// TwinCAT 3 PLC project Tc_SortingStation
// ProgramVersion: 3.1.4024.0
// libraries:
//   PlantControl and CMs, * (ArmAutomation)
//   Tc2_Standard, * (Beckhoff Automation GmbH)
//   Tc2_System, * (Beckhoff Automation GmbH)
//   Tc3_Module, * (Beckhoff Automation GmbH)
// project tree:
//   DUTs/ CM_DIN_UDT.TcDUT, CM_DO_UDT.TcDUT, CM_Vision_UDT.TcDUT
//   GVLs/ FIO.TcGVL, GVL.TcGVL
//   / PlcTask.TcTTO
//   POUs/ControlModules/ CM_DIN.TcPOU, CM_DO.TcPOU, CM_VisionSensor.TcPOU
//   POUs/EquipmentModules/FBD/ FB_ConveyorEntry_FBD.TcPOU
//   POUs/EquipmentModules/LAD/ FB_Conveyor.TcPOU, FB_Sorter.TcPOU
//   POUs/EquipmentModules/ST/ FB_ConveyorEntry_ST.TcPOU, FB_ConveyorExit_ST.TcPOU
//   POUs/ MAIN.TcPOU
// real-time tasks:
//   TASK PlcTask: cycle T#10ms, priority 20, ADS port 350

CONFIGURATION Tc_SortingStation
    RESOURCE PLC ON TwinCAT3
        TASK PlcTask(INTERVAL := T#10ms, PRIORITY := 20);
        PROGRAM MAIN WITH PlcTask : MAIN;
    END_RESOURCE
END_CONFIGURATION

// ---- DUTs/CM_DIN_UDT.TcDUT
TYPE CM_DIN_UDT :
STRUCT
	SensorInput : BOOL;
	
	AutoHigh : BOOL;
END_STRUCT
END_TYPE

// ---- DUTs/CM_DO_UDT.TcDUT
TYPE CM_DO_UDT :
STRUCT
	PI_Enable : BOOL;
	
	PO_HighCommand : BOOL;
	PO_LowCommand : BOOL;
END_STRUCT
END_TYPE

// ---- DUTs/CM_Vision_UDT.TcDUT
TYPE CM_Vision_UDT :
STRUCT
	Input : DINT;
	
	PO_PV : DINT;
END_STRUCT
END_TYPE

// ---- GVLs/FIO.TcGVL
{attribute 'qualified_only'}
VAR_GLOBAL

//Sensor	Bool	FACTORY I/O (Running)	496	FALSE
//Sensor	Bool	FACTORY I/O (Paused)	497	FALSE
//Sensor	Bool	FACTORY I/O (Reset)	498	FALSE
bAtExit : BOOL;	//Sensor	Bool	At exit	2	TRUE

//bEmgStop : BOOL; //Sensor	Bool	Emergency stop	0	TRUE
//bStart : BOOL;	//Sensor	Bool	Start	1	FALSE
//bStop : BOOL;	//Sensor	Bool	Stop	3	TRUE
//bReset : BOOL;	//Sensor	Bool	Reset	4	FALSE
//bManual : BOOL;	//Sensor	Bool	Manual	5	TRUE
//bAuto : BOOL; 	//Sensor	Bool	Auto	6	FALSE

//Sensor	Float	FACTORY I/O (Time Scale)	240	0
iVisionSensor : DINT;	//Sensor	Int	Vision sensor	0	0
//Actuator	Bool	FACTORY I/O (Run)	496	FALSE
//Actuator	Bool	FACTORY I/O (Pause)	497	FALSE
//Actuator	Bool	FACTORY I/O (Reset)	498	FALSE
bEmitter : BOOL; //Actuator	Bool	Emitter	0	TRUE
bConveyorEntry_out: BOOL; 	//Actuator	Bool	Entry conveyor	1	FALSE
bConveyorExit_out : BOOL; 		//Actuator	Bool	Exit conveyor	2	FALSE
bStopBlade : BOOL; 	//Actuator	Bool	Stop blade	3	FALSE
//Actuator	Bool	-	6	FALSE
bSorter_1_out : BOOL;	//Actuator	Bool	Sorter 1 belt	5	FALSE
bSorter_1_turn : BOOL;	//Actuator	Bool	Sorter 1 turn	4	FALSE
//Actuator	Bool	-	9	FALSE
bSorter_2_out : BOOL;	//Actuator	Bool	Sorter 2 belt	8	FALSE
bSorter_2_turn : BOOL;	//Actuator	Bool	Sorter 2 turn	7	FALSE
//Actuator	Bool	-	12	FALSE
bSorter_3_out : BOOL;	//Actuator	Bool	Sorter 3 belt	11	FALSE
bSorter_3_turn : BOOL;	//Actuator	Bool	Sorter 3 turn	10	FALSE
//Actuator	Bool	Remover 1	13	TRUE
//Actuator	Bool	Remover 2	14	TRUE
//Actuator	Bool	Remover 3	15	TRUE
//Actuator	Bool	Start light	16	FALSE
//Actuator	Bool	Stop light	17	FALSE
//Actuator	Bool	Reset light	18	FALSE
//Actuator	Int	FACTORY I/O (Camera Position)	240	0
//Actuator	Int	Counter 3	2	0
//Actuator	Int	Counter 1	0	0
//Actuator	Int	Counter 2	1	0

END_VAR

// ---- GVLs/GVL.TcGVL
{attribute 'qualified_only'}
VAR_GLOBAL
	GREEN_BOTTOM : BOOL; // 4
	GREEN_TOP : BOOL;	// 5
	GREEN_MIDDLE : BOOL; // 6
	
	BLUE_BOTTOM : BOOL; // 1
	BLUE_TOP : BOOL; // 2
	BLUE_MIDDLE : BOOL; // 3
	
	SortingDone : BOOL;
	readyForSorting : BOOL;
END_VAR

// ---- POUs/MAIN.TcPOU
PROGRAM MAIN
VAR
	
	//FBs
	fbPlantControl : PlantAndCMs.FB_PlantControl_mode_1;
	Ctrl_data_Plant : PlantAndCMs.Udt_PlantControl_Mode_1;
	
	//Equipment modules structured IN LADDER
	LAD_fbConveyorEntry : FB_Conveyor;
	LAD_fbSorter : FB_Sorter;
	
	//Equipment modules structured in ST
	ST_fbConveyorEntry : FB_ConveyorEntry_ST;
	ST_fbConveyorExit : FB_ConveyorExit_ST;
	
	// Control modules call
	cmVision : CM_VisionSensor;
	Ctrl_data_vision : CM_Vision_UDT;
	
	cmConveyor1 : CM_DO;
	cmConveyor2 : CM_DO;
	Ctrl_data_Conveyor1 : CM_DO_UDT;
	Ctrl_data_Conveyor2 : CM_DO_UDT;
	
	cmAtExit : CM_DIN;
	Ctrl_data_exit : CM_DIN_UDT;
	
	cmSorter1 : CM_DO;
	Crtl_data_sorter1 : CM_DO_UDT;
	cmSorter2 : CM_DO;
	Crtl_data_sorter2 : CM_DO_UDT;
	cmSorter3 : CM_DO;
	Crtl_data_sorter3 : CM_DO_UDT;
	
	cmStopBlade : CM_DO;
	crtl_data_StopBlade : CM_DO_UDT;
	
	cmEmitter : CM_DO;
	ctrl_data_emitter : CM_DO_UDT;
	
END_VAR

VAR_IN_OUT
	
END_VAR



fbPlantControl(
	on_in := TRUE,
	Auto_In := PlantAndCMs.FIO.bAuto,
	Manual_In := PlantAndCMs.FIO.bManual,
	
	EmgStop_In := PlantAndCMs.FIO.bEmgStop,
	Start_In := PlantAndCMs.FIO.bStart,
	Stop_In := PlantAndCMs.FIO.bStop, 
	Reset_In := PlantAndCMs.FIO.bReset,
	
	Ctrl_Plant := Ctrl_data_Plant
);
	

LAD_fbConveyorEntry(
		control_data := Ctrl_data_plant,
		
		control_data_vision := Ctrl_data_vision,
		control_data_Conveyor1 := Ctrl_data_Conveyor1,
		control_data_StopBlade := crtl_data_StopBlade,
		control_data_emitter := ctrl_data_emitter
		);	
	
LAD_fbSorter(
		control_data := Ctrl_data_plant,
		control_data_vision := Ctrl_data_vision,
		control_data_Conveyor2 := Ctrl_data_Conveyor2,
		control_data_sorter1 := Crtl_data_sorter1,
		control_data_sorter2 := Crtl_data_sorter2,
		control_data_sorter3 := Crtl_data_sorter3,
		control_data_atExit := Ctrl_data_exit,
	
	);	

(*
ST_fbConveyorEntry(
		control_data := Ctrl_data_plant,
		
		control_data_vision := Ctrl_data_vision,
		control_data_Conveyor1 := Ctrl_data_Conveyor1,
		control_data_StopBlade := crtl_data_StopBlade,
		control_data_emitter := ctrl_data_emitter
		);	

ST_fbConveyorExit(
		control_data := Ctrl_data_plant,
		control_data_vision := Ctrl_data_vision,
		control_data_Conveyor2 := Ctrl_data_Conveyor2,
		control_data_sorter1 := Crtl_data_sorter1,
		control_data_sorter2 := Crtl_data_sorter2,
		control_data_sorter3 := Crtl_data_sorter3,
		control_data_atExit := Ctrl_data_exit
		);
*)
		

//// CM Calls
cmConveyor1( 
	Control_data_DO := Ctrl_data_Conveyor1,
	
   	PO_HighCommand => FIO.bConveyorEntry_out
	); 
 
cmConveyor2(
	Control_data_DO := Ctrl_data_Conveyor2,
	PO_HighCommand => FIO.bConveyorExit_out
	);
	
cmAtExit(
	PI_autoHigh := FIO.bAtExit,
	Control_data := Ctrl_data_exit);

	
cmVision(
	SensorInput := FIO.iVisionSensor,
	control_data_vision := Ctrl_data_Vision);
	
cmSorter1(
	Control_data_DO := Crtl_data_sorter1,
	PO_HighCommand => FIO.bSorter_1_out, 
	PO_HighCommand => FIO.bSorter_1_turn
	);
cmSorter2(
	Control_data_DO := Crtl_data_sorter2,
	PO_HighCommand => FIO.bSorter_2_out, 
	PO_HighCommand => FIO.bSorter_2_turn
	);
	
cmSorter3(
	Control_data_DO := Crtl_data_sorter3,
	PO_HighCommand => FIO.bSorter_3_out,
	PO_HighCommand => FIO.bSorter_3_turn
	);
	
cmStopBlade(
	Control_data_DO := crtl_data_StopBlade,
	PO_HighCommand => FIO.bStopBlade
	);
cmEmitter(
	PO_HighCommand => FIO.bEmitter,
	Control_data_DO := ctrl_data_emitter
	);

END_PROGRAM

// ---- POUs/EquipmentModules/LAD/FB_Conveyor.TcPOU
FUNCTION_BLOCK FB_Conveyor
VAR_INPUT
	
END_VAR
VAR_OUTPUT
END_VAR
VAR
	on : BOOL;
	timer0_emitter : Tc2_Standard.TP;
	EmitterTrigger : BOOL;
	Timer1 : Tc2_Standard.TON;
	Step_0_Standby : BOOL;
	Step_1 : BOOL;
	Step_2 : BOOL;
	Step_3 : BOOL;
	Step_4 : BOOL;
	Step_5 : BOOL;
	Step_6 : BOOL;
	Step_7 : BOOL;
	Step_10 : BOOL;
	Step_15 : BOOL;
	step_last : BOOL;
	
	condition : BOOL;
	
	Opstart_puls_OS : BOOL;

	
	Initialiser_SQ: BOOL;
END_VAR
VAR_IN_OUT
	control_data : PlantAndCMs.Udt_PlantControl_Mode_1;
	
	control_data_vision : CM_Vision_UDT;
	control_data_Conveyor1 : CM_DO_UDT;
	
	control_data_StopBlade : CM_DO_UDT;
	control_data_emitter : CM_DO_UDT;
END_VAR
VAR // added by the converter: edge detectors and wires of the graphical bodies
    _w1, _w2, _w3, _w4, _w5, _w6, _w7, _w8, _w9, _w10, _w11, _w12, _w13, _w14, _w15, _w16, _w17 : BOOL;
END_VAR

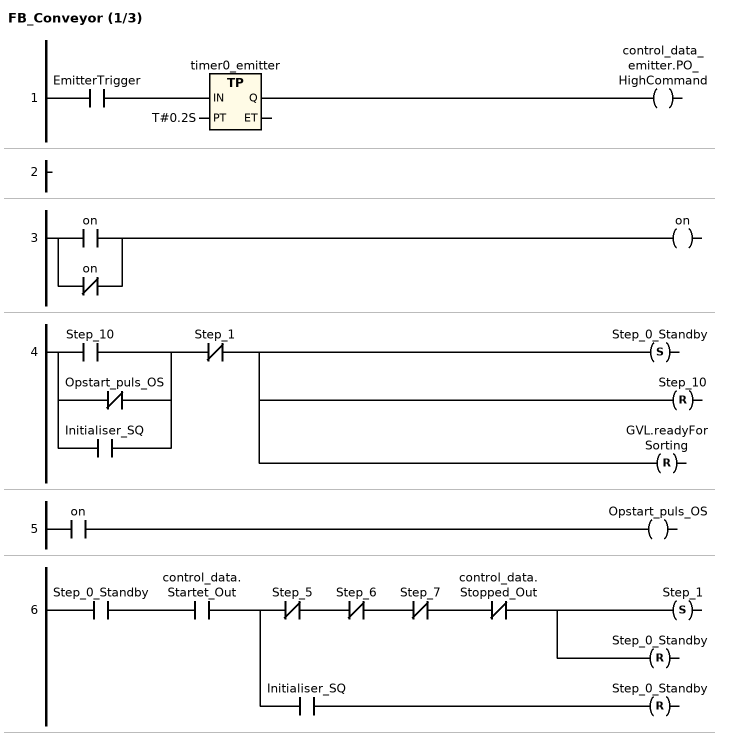
// NETWORK 1
timer0_emitter(IN := EmitterTrigger, PT := T#0.2S); // TP
control_data_emitter.PO_HighCommand := timer0_emitter.Q;

// NETWORK 2

// NETWORK 3
on := on OR NOT on;

// NETWORK 4
_w1 := (Step_10 OR NOT Opstart_puls_OS OR Initialiser_SQ) AND NOT Step_1;
Step_0_Standby S= _w1;
Step_10 R= _w1;
GVL.readyForSorting R= _w1;

// NETWORK 5
Opstart_puls_OS := on;

// NETWORK 6
_w2 := Step_0_Standby AND control_data.Startet_Out;
_w3 := _w2 AND NOT Step_5 AND NOT Step_6 AND NOT Step_7 AND NOT control_data.Stopped_Out;
Step_1 S= _w3;
Step_0_Standby R= _w3;
Step_0_Standby R= _w2 AND Initialiser_SQ;

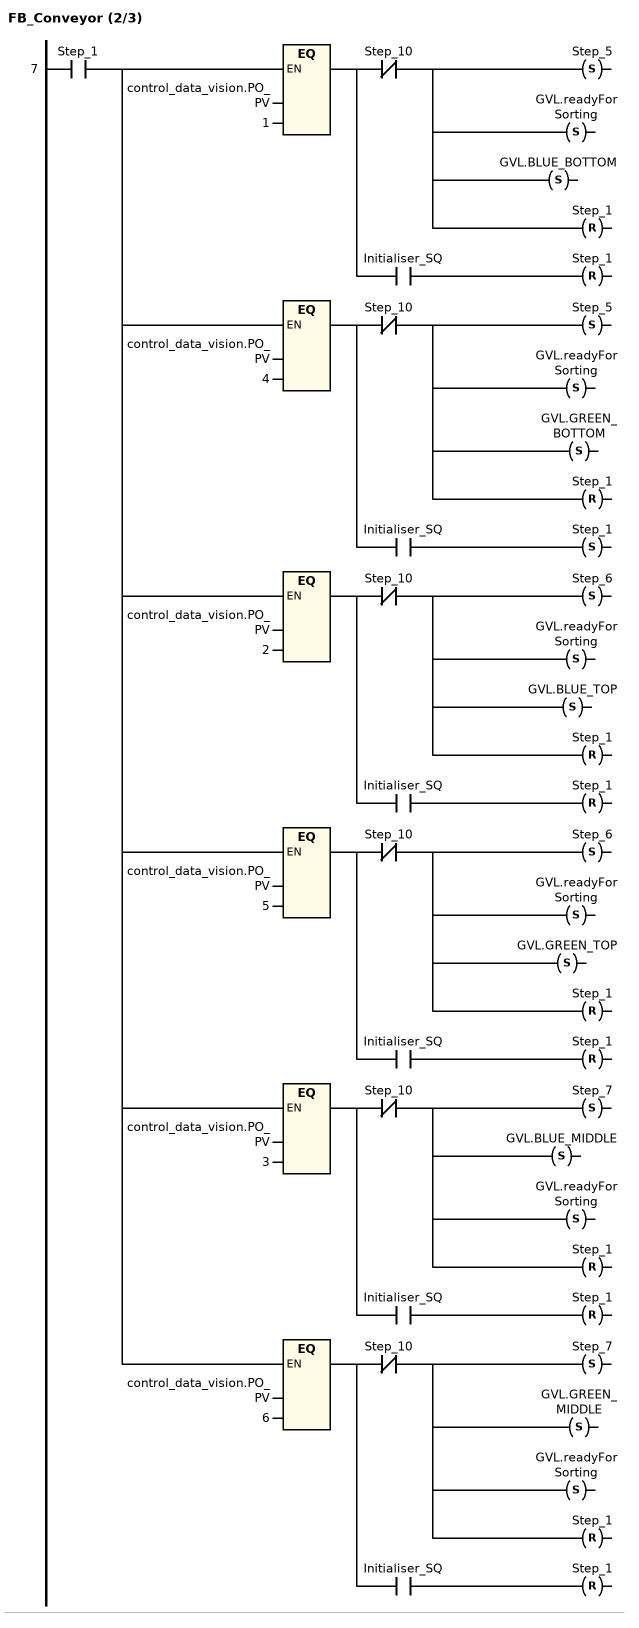
// NETWORK 7
_w4 := Step_1;
_w5 := _w4 AND control_data_vision.PO_PV = 1;
_w6 := _w5 AND NOT Step_10;
Step_5 S= _w6;
GVL.readyForSorting S= _w6;
GVL.BLUE_BOTTOM S= _w6;
Step_1 R= _w6;
Step_1 R= _w5 AND Initialiser_SQ;
_w7 := _w4 AND control_data_vision.PO_PV = 4;
_w8 := _w7 AND NOT Step_10;
Step_5 S= _w8;
GVL.readyForSorting S= _w8;
GVL.GREEN_BOTTOM S= _w8;
Step_1 R= _w8;
Step_1 S= _w7 AND Initialiser_SQ;
_w9 := _w4 AND control_data_vision.PO_PV = 2;
_w10 := _w9 AND NOT Step_10;
Step_6 S= _w10;
GVL.readyForSorting S= _w10;
GVL.BLUE_TOP S= _w10;
Step_1 R= _w10;
Step_1 R= _w9 AND Initialiser_SQ;
_w11 := _w4 AND control_data_vision.PO_PV = 5;
_w12 := _w11 AND NOT Step_10;
Step_6 S= _w12;
GVL.readyForSorting S= _w12;
GVL.GREEN_TOP S= _w12;
Step_1 R= _w12;
Step_1 R= _w11 AND Initialiser_SQ;
_w13 := _w4 AND control_data_vision.PO_PV = 3;
_w14 := _w13 AND NOT Step_10;
Step_7 S= _w14;
GVL.BLUE_MIDDLE S= _w14;
GVL.readyForSorting S= _w14;
Step_1 R= _w14;
Step_1 R= _w13 AND Initialiser_SQ;
_w15 := _w4 AND control_data_vision.PO_PV = 6;
_w16 := _w15 AND NOT Step_10;
Step_7 S= _w16;
GVL.GREEN_MIDDLE S= _w16;
GVL.readyForSorting S= _w16;
Step_1 R= _w16;
Step_1 R= _w15 AND Initialiser_SQ;

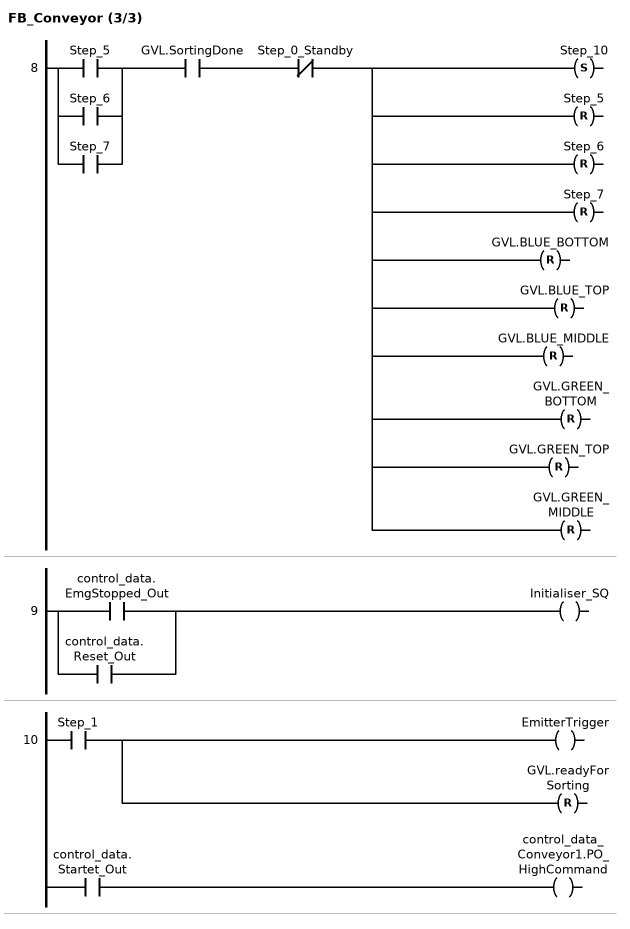
// NETWORK 8
_w17 := (Step_5 OR Step_6 OR Step_7) AND GVL.SortingDone AND NOT Step_0_Standby;
Step_10 S= _w17;
Step_5 R= _w17;
Step_6 R= _w17;
Step_7 R= _w17;
GVL.BLUE_BOTTOM R= _w17;
GVL.BLUE_TOP R= _w17;
GVL.BLUE_MIDDLE R= _w17;
GVL.GREEN_BOTTOM R= _w17;
GVL.GREEN_TOP R= _w17;
GVL.GREEN_MIDDLE R= _w17;

// NETWORK 9
Initialiser_SQ := control_data.EmgStopped_Out OR control_data.Reset_Out;

// NETWORK 10
EmitterTrigger := Step_1;
GVL.readyForSorting R= Step_1;
control_data_Conveyor1.PO_HighCommand := control_data.Startet_Out;

END_FUNCTION_BLOCK

// ---- POUs/EquipmentModules/LAD/FB_Sorter.TcPOU
FUNCTION_BLOCK FB_Sorter
VAR_INPUT
END_VAR
VAR_OUTPUT
END_VAR
VAR
	on : BOOL;
	
	rTrigAtExit : Tc2_Standard.R_TRIG;
	exitTrigger : BOOL;
	atExitEdgeDetected : BOOL;
	
	Step_0_Standby : BOOL;
	Step_1 : BOOL;
	Step_2 : BOOL;
	Step_3 : BOOL;
	Step_4 : BOOL;
	Step_5 : BOOL;
	Step_6 : BOOL;
	Step_7 : BOOL;
	Step_10 : BOOL;
	Step_15 : BOOL;
	step_last : BOOL;
	
	dummy : BOOL;
	
	condition : BOOL;
	
	Opstart_puls_OS : BOOL;

	Initialiser_SQ: BOOL;
END_VAR
VAR_IN_OUT
	control_data : PlantAndCMs.Udt_PlantControl_Mode_1;
	
	control_data_vision : CM_Vision_UDT;
	control_data_Conveyor2 : CM_DO_UDT;
	
	control_data_sorter1 : CM_DO_UDT;
	control_data_sorter2 : CM_DO_UDT;
	control_data_sorter3 : CM_DO_UDT;
	
	control_data_atExit : CM_DIN_UDT;
	
	
END_VAR
VAR // added by the converter: edge detectors and wires of the graphical bodies
    _w1, _w2, _w3, _w4, _w5, _w6, _w7, _w8, _w9, _w10, _w11 : BOOL;
END_VAR

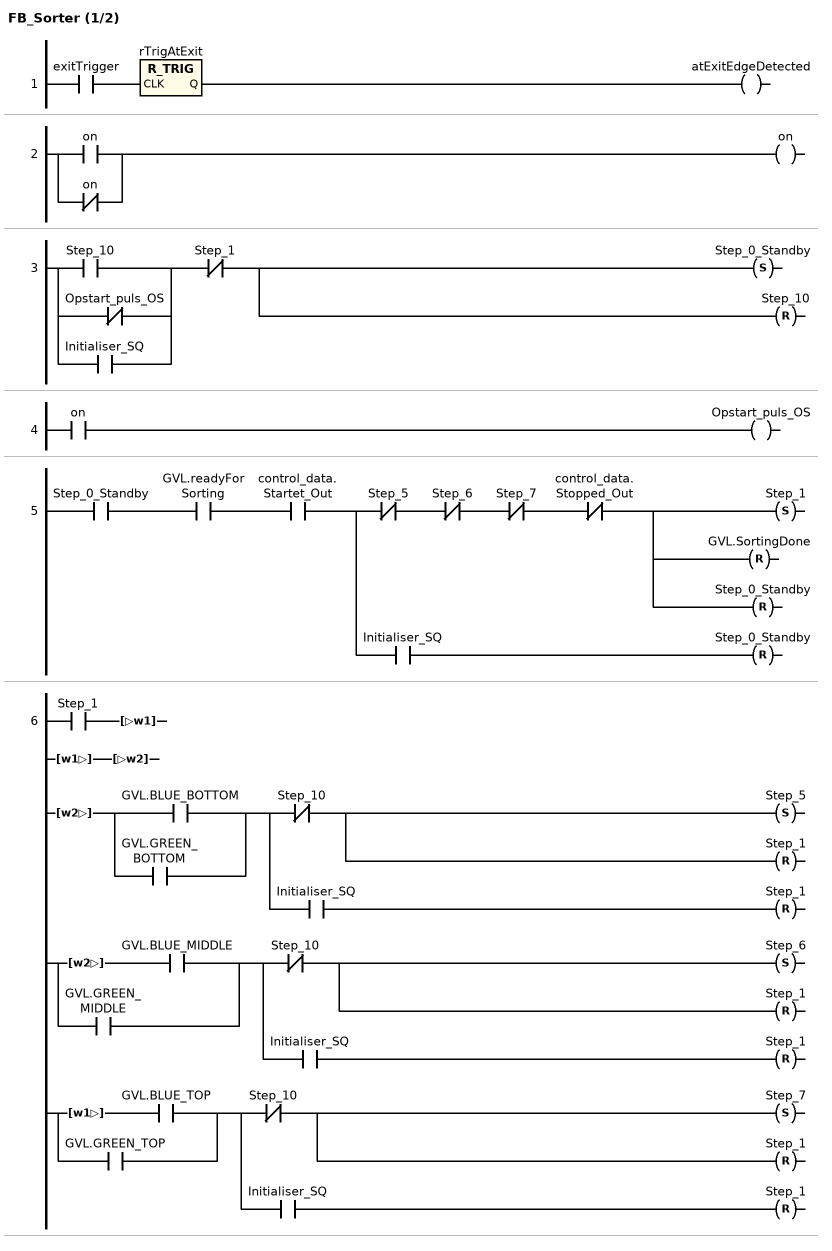
// NETWORK 1
rTrigAtExit(CLK := exitTrigger); // R_TRIG
atExitEdgeDetected := rTrigAtExit.Q;

// NETWORK 2
on := on OR NOT on;

// NETWORK 3
_w1 := (Step_10 OR NOT Opstart_puls_OS OR Initialiser_SQ) AND NOT Step_1;
Step_0_Standby S= _w1;
Step_10 R= _w1;

// NETWORK 4
Opstart_puls_OS := on;

// NETWORK 5
_w2 := Step_0_Standby AND GVL.readyForSorting AND control_data.Startet_Out;
_w3 := _w2 AND NOT Step_5 AND NOT Step_6 AND NOT Step_7 AND NOT control_data.Stopped_Out;
Step_1 S= _w3;
GVL.SortingDone R= _w3;
Step_0_Standby R= _w3;
Step_0_Standby R= _w2 AND Initialiser_SQ;

// NETWORK 6
_w4 := Step_1;
_w5 := _w4 AND (GVL.BLUE_BOTTOM OR GVL.GREEN_BOTTOM);
_w6 := _w5 AND NOT Step_10;
Step_5 S= _w6;
Step_1 R= _w6;
Step_1 R= _w5 AND Initialiser_SQ;
_w7 := _w4 AND GVL.BLUE_MIDDLE OR GVL.GREEN_MIDDLE;
_w8 := _w7 AND NOT Step_10;
Step_6 S= _w8;
Step_1 R= _w8;
Step_1 R= _w7 AND Initialiser_SQ;
_w9 := _w4 AND GVL.BLUE_TOP OR GVL.GREEN_TOP;
_w10 := _w9 AND NOT Step_10;
Step_7 S= _w10;
Step_1 R= _w10;
Step_1 R= _w9 AND Initialiser_SQ;

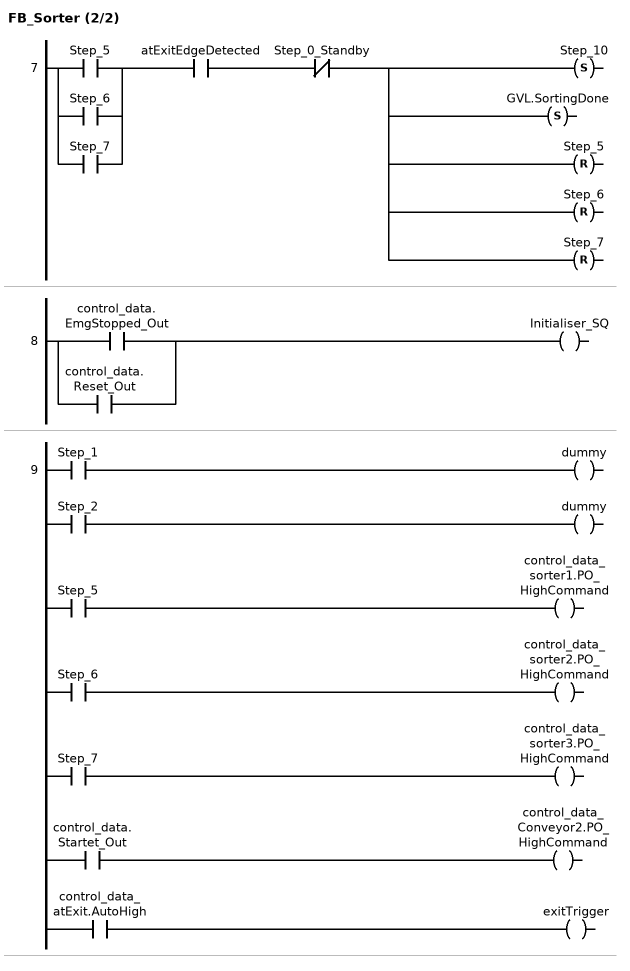
// NETWORK 7
_w11 := (Step_5 OR Step_6 OR Step_7) AND atExitEdgeDetected AND NOT Step_0_Standby;
Step_10 S= _w11;
GVL.SortingDone S= _w11;
Step_5 R= _w11;
Step_6 R= _w11;
Step_7 R= _w11;

// NETWORK 8
Initialiser_SQ := control_data.EmgStopped_Out OR control_data.Reset_Out;

// NETWORK 9
dummy := Step_1;
dummy := Step_2;
control_data_sorter1.PO_HighCommand := Step_5;
control_data_sorter2.PO_HighCommand := Step_6;
control_data_sorter3.PO_HighCommand := Step_7;
control_data_Conveyor2.PO_HighCommand := control_data.Startet_Out;
exitTrigger := control_data_atExit.AutoHigh;

END_FUNCTION_BLOCK

// ---- POUs/EquipmentModules/ST/FB_ConveyorEntry_ST.TcPOU
FUNCTION_BLOCK FB_ConveyorEntry_ST
VAR_INPUT
END_VAR
VAR_OUTPUT
END_VAR
VAR
	step : INT;
	RtrigInitTrigger : R_TRIG;
	initTrigger : BOOL := TRUE;
	
	eMitterTimer : Tc2_Standard.TP;
	startEmitting : BOOL;
	
END_VAR
VAR_IN_OUT
	control_data : PlantAndCMs.Udt_PlantControl_Mode_1;
	
	control_data_vision : CM_Vision_UDT;
	control_data_Conveyor1 : CM_DO_UDT;
	
	control_data_StopBlade : CM_DO_UDT;
	control_data_emitter : CM_DO_UDT;
END_VAR

RtrigInitTrigger(CLK :=initTrigger);

eMitterTimer(IN := StartEmitting, pt := T#0.2S);


CASE step OF 
	0 : // Init
	
		IF control_data.Auto_Out THEN
			initTrigger := FALSE;
			step := 1;
		END_IF
	
	1: // Step 1 start machine
		
		IF control_data.Startet_Out THEN
			initTrigger := TRUE;
			step := 2;
		END_IF
	2:			
		
		IF control_data_vision.PO_PV = 0 THEN
			startEmitting := TRUE;
			step := 5;
		END_IF
	
	5: 
		startEmitting := FALSE;
		GVL.readyForSorting := FALSE;
		GVL.SortingDone := FALSE;
		
		IF control_data_vision.PO_PV = 1 THEN
			GVL.BLUE_TOP := TRUE;
			GVL.BLUE_BOTTOM := FALSE;
			GVL.BLUE_MIDDLE := FALSE;
			GVL.GREEN_TOP := FALSE;
			GVL.GREEN_BOTTOM := FALSE;
			GVL.GREEN_MIDDLE := FALSE;
			step := 11;
		END_IF
		IF control_data_vision.PO_PV = 2 THEN
			GVL.BLUE_TOP := FALSE;
			GVL.BLUE_BOTTOM := TRUE;
			GVL.BLUE_MIDDLE := FALSE;
			GVL.GREEN_TOP := FALSE;
			GVL.GREEN_BOTTOM := FALSE;
			GVL.GREEN_MIDDLE := FALSE;
			step := 11;
		END_IF
		IF control_data_vision.PO_PV = 3 THEN
			GVL.BLUE_TOP := FALSE;
			GVL.BLUE_BOTTOM := FALSE;
			GVL.BLUE_MIDDLE := TRUE;
			GVL.GREEN_TOP := FALSE;
			GVL.GREEN_BOTTOM := FALSE;
			GVL.GREEN_MIDDLE := FALSE;
			step := 11;
		END_IF
		IF control_data_vision.PO_PV = 4 THEN
			GVL.BLUE_TOP := FALSE;
			GVL.BLUE_BOTTOM := FALSE;
			GVL.BLUE_MIDDLE := FALSE;
			GVL.GREEN_TOP := TRUE;
			GVL.GREEN_BOTTOM := FALSE;
			GVL.GREEN_MIDDLE := FALSE;
			step := 11;
		END_IF
		IF control_data_vision.PO_PV = 5 THEN
			GVL.BLUE_TOP := FALSE;
			GVL.BLUE_BOTTOM := FALSE;
			GVL.BLUE_MIDDLE := FALSE;
			GVL.GREEN_TOP := FALSE;
			GVL.GREEN_BOTTOM := TRUE;
			GVL.GREEN_MIDDLE := FALSE;
			step := 11;
		END_IF
		IF control_data_vision.PO_PV = 6 THEN
			GVL.BLUE_TOP := FALSE;
			GVL.BLUE_BOTTOM := FALSE;
			GVL.BLUE_MIDDLE := FALSE;
			GVL.GREEN_TOP := FALSE;
			GVL.GREEN_BOTTOM := FALSE;
			GVL.GREEN_MIDDLE := TRUE;
			step := 11;
		END_IF
		

	11:
		GVL.readyForSorting := TRUE;
		
		IF GVL.SortingDone THEN
			GVL.BLUE_TOP := FALSE;
			GVL.BLUE_BOTTOM := FALSE;
			GVL.BLUE_MIDDLE := FALSE;
			GVL.GREEN_TOP := FALSE;
			GVL.GREEN_BOTTOM := FALSE;
			GVL.GREEN_MIDDLE := FALSE;
			
			startEmitting := TRUE;
			
			step := 2;
		END_IF
		
END_CASE


control_data_emitter.PO_HighCommand := eMitterTimer.Q;

control_data_Conveyor1.PO_HighCommand := control_data.Startet_Out;

END_FUNCTION_BLOCK

// ---- POUs/EquipmentModules/ST/FB_ConveyorExit_ST.TcPOU
FUNCTION_BLOCK FB_ConveyorExit_ST
VAR_INPUT
END_VAR
VAR_OUTPUT
END_VAR
VAR
	rTrigExit : Tc2_Standard.R_TRIG;
	ExitTrigger : BOOL;
	ExitEdgeDetected : BOOL;
	
	step : INT;
END_VAR
VAR_IN_OUT
	control_data : PlantAndCMs.Udt_PlantControl_Mode_1;
	
	control_data_vision : CM_Vision_UDT;
	control_data_Conveyor2 : CM_DO_UDT;
	
	control_data_sorter1 : CM_DO_UDT;
	control_data_sorter2 : CM_DO_UDT;
	control_data_sorter3 : CM_DO_UDT;
	
	control_data_atExit : CM_DIN_UDT;
END_VAR

rTrigExit(CLK := ExitTrigger, Q => ExitEdgeDetected);

CASE step OF 
	0 : // Init
	IF control_data.Auto_Out AND control_data.Startet_Out THEN
		step := 1;
	END_IF
	
	1: // wait for ready signal from ceonveyor entry
	
	
	IF GVL.readyForSorting THEN
		step := 2;
	END_IF
	
	2 : // check for GVL. which brick and act accordingly
	IF GVL.BLUE_TOP OR GVL.GREEN_TOP THEN
		step := 5;
	ELSIF GVL.BLUE_MIDDLE OR GVL.GREEN_MIDDLE THEN
		step := 10;
	ELSIF GVL.GREEN_BOTTOM OR GVL.BLUE_BOTTOM THEN
		step := 15;
		
	END_IF
	
	5:
		GVL.BLUE_TOP := FALSE;
		GVL.BLUE_BOTTOM := FALSE;
		GVL.BLUE_MIDDLE := FALSE;
		GVL.GREEN_TOP := FALSE;
		GVL.GREEN_BOTTOM := FALSE;
		GVL.GREEN_MIDDLE := FALSE;
		IF ExitEdgeDetected THEN
			step := 1;
			GVL.SortingDone := TRUE;
		END_IF
	10:
		GVL.BLUE_TOP := FALSE;
		GVL.BLUE_BOTTOM := FALSE;
		GVL.BLUE_MIDDLE := FALSE;
		GVL.GREEN_TOP := FALSE;
		GVL.GREEN_BOTTOM := FALSE;
		GVL.GREEN_MIDDLE := FALSE;
		IF ExitEdgeDetected THEN
			step := 1;
			GVL.SortingDone := TRUE;
		END_IF
	15:
		GVL.BLUE_TOP := FALSE;
		GVL.BLUE_BOTTOM := FALSE;
		GVL.BLUE_MIDDLE := FALSE;
		GVL.GREEN_TOP := FALSE;
		GVL.GREEN_BOTTOM := FALSE;
		GVL.GREEN_MIDDLE := FALSE;
		IF ExitEdgeDetected THEN
			step := 1;
			GVL.SortingDone := TRUE;
		END_IF
	 
END_CASE

ExitTrigger := control_data_atExit.AutoHigh; 

control_data_Sorter1.PO_HighCommand := step = 5;
control_data_sorter2.PO_HighCommand := step = 10;
control_data_sorter3.PO_HighCommand := step = 15;

control_data_Conveyor2.PO_HighCommand := step = 5 OR step = 10 OR step = 15;

END_FUNCTION_BLOCK

// ---- POUs/ControlModules/CM_VisionSensor.TcPOU
FUNCTION_BLOCK CM_VisionSensor
VAR_INPUT
	SensorInput : DINT;
END_VAR
VAR_OUTPUT
	SensorOutput : DINT;
END_VAR
VAR_IN_OUT
	control_data_vision : CM_Vision_UDT;
END_VAR


SensorOutput := SensorInput;

control_data_vision.PO_PV := SensorOutput;

END_FUNCTION_BLOCK

// ---- POUs/ControlModules/CM_DO.TcPOU
FUNCTION_BLOCK CM_DO
VAR_INPUT
	PI_Enable : BOOL;
END_VAR
VAR_OUTPUT
	PO_HighCommand : BOOL;
	PO_LowCommand : BOOL;
END_VAR
VAR_IN_OUT
	Control_data_DO : CM_DO_UDT;
END_VAR

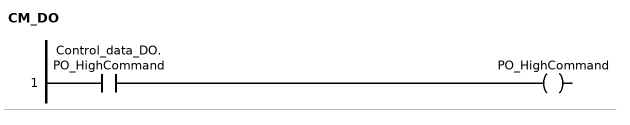
// NETWORK 1
PO_HighCommand := Control_data_DO.PO_HighCommand;

END_FUNCTION_BLOCK

// ---- POUs/ControlModules/CM_DIN.TcPOU
FUNCTION_BLOCK CM_DIN
VAR_INPUT
	PI_autoHigh : BOOL;
END_VAR
VAR_OUTPUT
END_VAR
VAR_IN_OUT
	Control_data : CM_DIN_UDT;
END_VAR

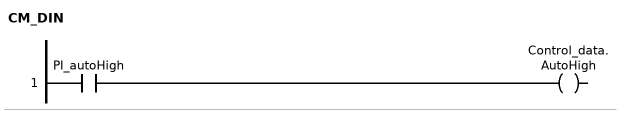
// NETWORK 1
Control_data.AutoHigh := PI_autoHigh;

END_FUNCTION_BLOCK

// ---- POUs/EquipmentModules/FBD/FB_ConveyorEntry_FBD.TcPOU
FUNCTION_BLOCK FB_ConveyorEntry_FBD
VAR_INPUT
END_VAR
VAR_OUTPUT
END_VAR
VAR
	
	timer0_emitter : Tc2_Standard.TP;
	EmitterTrigger : BOOL;
	Timer1 : Tc2_Standard.TON;
	Step_0_Standby : BOOL;
	Step_1 : BOOL;
	Step_2 : BOOL;
	Step_3 : BOOL;
	Step_4 : BOOL;
	Step_5 : BOOL;
	Step_6 : BOOL;
	Step_7 : BOOL;
	Step_10 : BOOL;
	Step_15 : BOOL;
	step_last : BOOL;
	
	condition : BOOL;
	
	Opstart_puls_OS : BOOL;

	
	Initialiser_SQ: BOOL;
END_VAR
VAR_IN_OUT
	control_data : PlantAndCMs.Udt_PlantControl_Mode_1;
	
	control_data_vision : CM_Vision_UDT;
	control_data_Conveyor1 : CM_DO_UDT;
	
	control_data_StopBlade : CM_DO_UDT;
	control_data_emitter : CM_DO_UDT;
END_VAR

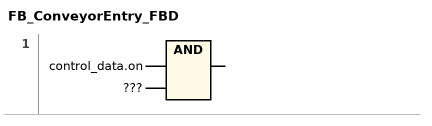
// NETWORK 1
(* control_data.on AND ???; result not used *)

END_FUNCTION_BLOCK
